TYPE ST_P_GET_OP_STATE :
STRUCT
	CheckState:				BOOL;
	OperationName:			STRING;
	OperationIndex:			INT;
	Barcode:				INT;
END_STRUCT
END_TYPE

(* stored: Version 1.1.0.1, ProductVersion 3.1.4024.10
   DUT ST_P_GET_OP_STATE: Id {9de30d1d-fa8b-4ec8-93e8-a4faa34748bb} *)
